FUNCTION_BLOCK EcMasterGetDeviceState IMPLEMENTS IEcTask
VAR_INPUT
END_VAR
VAR_OUTPUT
END_VAR
VAR
	iState : INT;
	getDeviceState : Tc2_EtherCAT.FB_EcGetSlaveState;
	_execute: BOOL;
	_done: BOOL;
	_busy: BOOL;
	_error: BOOL;
	_netId: AMSNETID;
END_VAR

CASE iState OF
	0:
		IF _execute THEN
			_done := FALSE;
			_busy := TRUE;
			_error := FALSE;
			getDeviceState.bExecute := TRUE;
			IF getDeviceState.bBusy THEN
				iState := 10;
				_execute := false;
			END_IF
		END_IF
	10:
		IF NOT getDeviceState.bBusy THEN
			IF NOT getDeviceState.bError THEN
				_done := TRUE;
			ELSE
				_error := TRUE;
			END_IF
			_busy := FALSE;
			getDeviceState.bExecute := FALSE;
			iState := 0;
		END_IF
END_CASE

getDeviceState(sNetId := Tc2_System.F_CreateAmsNetId(nIds := NetId));

{warning 'add method implementation '}
METHOD Abort : BOOL
getDeviceState.bExecute := FALSE;
_busy := FALSE;
_execute := FALSE;
Abort := TRUE;
iState := 0;
END_METHOD

{warning 'add property implementation'}
PROPERTY Busy : BOOL
GET
Busy := _busy;
END_GET
END_PROPERTY

PROPERTY DeviceAddr : uint
GET
DeviceAddr := getDeviceState.nSlaveAddr;
END_GET
SET
getDeviceState.nSlaveAddr := DeviceAddr;
END_SET
END_PROPERTY

PROPERTY DeviceState : ST_EcSlaveState
GET
DeviceState := getDeviceState.state;
END_GET
END_PROPERTY

{warning 'add property implementation'}
PROPERTY Done : BOOL
GET
Done := _done;
END_GET
END_PROPERTY

{warning 'add property implementation'}
PROPERTY Error : BOOL
GET
Error := _error;
END_GET
END_PROPERTY

{warning 'add method implementation '}
METHOD Execute : BOOL
IF NOT getDeviceState.bBusy THEN
	Execute := _execute := true;
END_IF
END_METHOD

{warning 'add property implementation'}
PROPERTY NetID : amsnetid
GET
NetID := _netId;
END_GET
SET
_netId := NetID;
END_SET
END_PROPERTY

END_FUNCTION_BLOCK

(* stored: Version 1.1.0.1, ProductVersion 3.1.4024.11
   POU EcMasterGetDeviceState: Id {5e1424d3-bf53-4170-a13e-7c1095e3c66d}, SpecialFunc None
   Method Abort: Id {abec5460-4ddc-46bf-8a99-853e0222d903}
   Property Busy: Id {dc62c4aa-f228-4b2d-b3e4-55add37f8b32}
   Get Get: Id {8b968973-541f-4cde-8942-8d1c826a1b0f}
   Property DeviceAddr: Id {15e138b0-2f3b-4e98-8d46-5d15aa60ca84}
   Get Get: Id {ae2feb77-bb28-4a09-aaee-30a0055aa7d5}
   Set Set: Id {e2f51ab3-dc0e-4c52-9581-4307d65c8247}
   Property DeviceState: Id {0012da42-ed8e-4c0e-9903-6e49a6305c48}
   Get Get: Id {1405ab92-ddc0-4014-8378-ebaa67d63c6e}
   Property Done: Id {bb03e3b1-3d15-408b-85bc-fe391e224ee3}
   Get Get: Id {2e48ea6c-6105-4b02-99ea-d7a5116d5bf4}
   Property Error: Id {34cc37aa-152a-492f-b545-353d17c45898}
   Get Get: Id {81c09089-73ac-4cd7-89f3-dd4ffc93650e}
   Method Execute: Id {c4a9273e-53df-49a5-bbc6-73d1c6473762}
   Property NetID: Id {b7976b66-bb9a-4cb7-9686-db9febffe9f6}
   Get Get: Id {cb9ca70f-d743-479a-8aaf-f075ba8ce2d3}
   Set Set: Id {65794dff-0f83-4592-a948-1dccd2b7177f} *)
